// SIMATIC STEP 7 (V5.x) project TEMPORIZADOR
// CPU: CPU 314C-2 DP
// station: Hardware
// station: TEMPO
// station: P_ADR_BUS
// program: Programa S7(1)

ORGANIZATION_BLOCK OB 1
TITLE = "Main Program Sweep (Cycle)"
VERSION : 0.1
VAR_TEMP
  OB1_EV_CLASS : BYTE ;	//Bits 0-3 = 1 (Coming event), Bits 4-7 = 1 (Event class 1)
  OB1_SCAN_1 : BYTE ;	//1 (Cold restart scan 1 of OB 1), 3 (Scan 2-n of OB 1)
  OB1_PRIORITY : BYTE ;	//Priority of OB Execution
  OB1_OB_NUMBR : BYTE ;	//1 (Organization block 1, OB1)
  OB1_RESERVED_1 : BYTE ;	//Reserved for system
  OB1_RESERVED_2 : BYTE ;	//Reserved for system
  OB1_PREV_CYCLE : INT ;	//Cycle time of previous OB1 scan (milliseconds)
  OB1_MIN_CYCLE : INT ;	//Minimum cycle time of OB1 (milliseconds)
  OB1_MAX_CYCLE : INT ;	//Maximum cycle time of OB1 (milliseconds)
  OB1_DATE_TIME : DATE_AND_TIME ;	//Date and time OB1 started
END_VAR
BEGIN
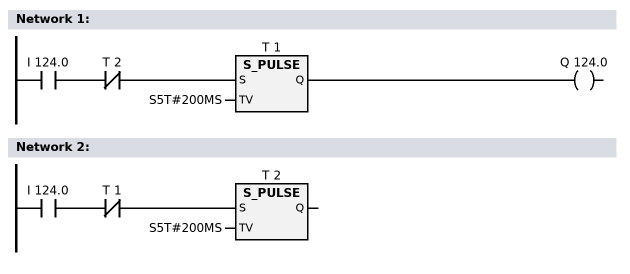
NETWORK
TITLE =
      A     I 124.0;
      AN    T 2;
      L     S5T#200MS;
      SP    T 1;
      NOP   0;
      NOP   0;
      NOP   0;
      A     T 1;
      =     Q 124.0;
NETWORK
TITLE =
      A     I 124.0;
      AN    T 1;
      L     S5T#200MS;
      SP    T 2;
      NOP   0;
      NOP   0;
      NOP   0;
      NOP   0;
END_ORGANIZATION_BLOCK
